FUNCTION Convert_DATE_TO_REAL : BOOL
VAR_INPUT
	in : DATE;
	out : REFERENCE TO REAL;
END_VAR
VAR
	converted : REAL;
END_VAR

converted := DATE_TO_REAL(in);

IF (REAL_TO_DATE(converted) <> in) THEN
	RETURN;
END_IF

out := converted;
Convert_DATE_TO_REAL := TRUE;

END_FUNCTION

(* stored: Version 1.1.0.1, ProductVersion 3.1.4024.12
   POU Convert_DATE_TO_REAL: Id {02c95f9e-8d6c-41d0-b1c6-7e1c4554fc46}, SpecialFunc None *)
